FUNCTION Convert_BYTE_TO_REAL : Hresult
VAR_INPUT
	in : BYTE;
	out : REFERENCE TO REAL;
END_VAR
VAR
	converted : REAL;
END_VAR
VAR CONSTANT
	INCOMPATIBLE : HRESULT := 16#9811070E;
END_VAR

converted := BYTE_TO_REAL(in);

IF (REAL_TO_BYTE(converted) <> in) THEN
	Convert_BYTE_TO_REAL := INCOMPATIBLE;
	RETURN;
END_IF

out := converted;

END_FUNCTION

(* stored: Version 1.1.0.1, ProductVersion 3.1.4024.12
   POU Convert_BYTE_TO_REAL: Id {f5723143-aba1-4154-8687-6be5c2bbef40}, SpecialFunc None *)
